FUNCTION_BLOCK TableDeserializer
VAR
	_DataString : POINTER TO STRING;
	dataLength : DINT;
	rowDefinition : __SYSTEM.AnyType;
	_RowCount : DINT;
	_ColumnDefinitionBuffer : ARRAY[0..MaxColumnCount - 1] OF __SYSTEM.AnyType;
	_ColumnNameBuffer : ARRAY[0..MaxColumnCount - 1] OF T_MaxString;
	columnNamesOutput : __SYSTEM.AnyType;
	definedColumns : INT;

	_Separator : STRING := ',';
	_NewLine : STRING := '$N'; // Default is Windows newline.
	_DecimalSeparator : STRING := '.';
END_VAR
VAR CONSTANT
	MaxColumnCount : INT := TableSerializationParameters.DeserializerMaxColumns;
	DefaultDecimalSeparator : STRING := '.';
END_VAR

{attribute 'monitoring' := 'call'}
PROPERTY DataString : POINTER TO STRING
GET
DataString := _DataString;
END_GET
SET
_DataString := DataString;
END_SET
END_PROPERTY

{attribute 'monitoring' := 'call'}
PROPERTY DecimalSeparator : STRING
GET
DecimalSeparator := _DecimalSeparator;
END_GET
SET
_DecimalSeparator := DecimalSeparator;
END_SET
END_PROPERTY

METHOD DefineColumnNamesOutput : REFERENCE TO TableDeserializer
VAR_INPUT
	columnNames : ANY; 
END_VAR
columnNamesOutput := columnNames;

DefineColumnNamesOutput REF= THIS^;
END_METHOD

METHOD DefineNextColumn : REFERENCE TO TableDeserializer
VAR_INPUT
	columnInFirstRow : ANY; 
END_VAR
IF (definedColumns < MaxColumnCount) THEN
	_ColumnDefinitionBuffer[definedColumns] := columnInFirstRow;
	definedColumns := definedColumns + 1;
END_IF

DefineNextColumn REF= THIS^;
END_METHOD

METHOD DefineRow : REFERENCE TO TableDeserializer
VAR_INPUT
	firstRow : ANY;
END_VAR
rowDefinition := firstRow;

DefineRow REF= THIS^;
END_METHOD

METHOD Deserialize : DINT
VAR_INPUT
	includingHeader : BOOL;
END_VAR
VAR
	caret : DINT;
END_VAR
dataLength := TO_DINT(LEN2(dataString));
IF (includingHeader) THEN
	caret := ReadHeader();
END_IF
caret := ReadAllRows(caret);

Deserialize := caret;
END_METHOD

{attribute 'monitoring' := 'call'}
PROPERTY NewLine : STRING
GET
NewLine := _NewLine;
END_GET
SET
_NewLine := NewLine;
END_SET
END_PROPERTY

METHOD PRIVATE ReadAllRows : DINT
VAR_INPUT
	startCaret : DINT;
END_VAR
VAR
	caret : DINT;
	i : DINT;
END_VAR
caret := startCaret;

FOR i := 0 TO _RowCount - 1 DO
	IF (caret >= dataLength) THEN
		EXIT;
	END_IF
	caret := ReadRow(i, caret);
END_FOR

ReadAllRows := caret;
END_METHOD

METHOD PRIVATE ReadHeader : DINT
VAR
	i : DINT;
	
	caret : DINT;
	lineEnd : DINT;
	cellLength : DINT;
	
	cell : T_MaxString;
END_VAR
ClearData(_ColumnNameBuffer);

lineEnd := TO_DINT(FIND2(pSrcString := _DataString, pFindString := ADR(_NewLine)));
IF (lineEnd = 0) THEN
	lineEnd := dataLength;
END_IF

FOR i := 0 TO definedColumns - 1 DO
	cellLength := TO_DINT(FIND2(pSrcString := _DataString + TO_DWORD(caret), pFindString := ADR(_Separator)));
	IF (caret + cellLength > lineEnd) THEN
		cellLength := lineEnd - caret;
	END_IF
	IF (cellLength = 0) THEN
		cellLength := lineEnd;
	END_IF

	MEMSET(destAddr := ADR(cell), fillByte := 0, n := SIZEOF(cell));
	MEMCPY(destAddr := ADR(cell), srcAddr := _DataString + TO_DWORD(caret), n := TO_UDINT(MIN(SIZEOF(cell) - 1, cellLength - 1)));
	StringToAny(cell, _ColumnNameBuffer[i]);
	
	IF (cellLength = dataLength) THEN
		caret := lineEnd;
	ELSIF (cellLength = lineEnd) THEN
		caret := lineEnd;
	ELSE
		caret := caret + cellLength;
	END_IF
END_FOR

MEMCPY(
	destAddr := columnNamesOutput.pValue,
	srcAddr := ADR(_ColumnNameBuffer),
	n := TO_UDINT(MIN(columnNamesOutput.diSize, SIZEOF(_ColumnNameBuffer)))
);

ReadHeader := caret;
END_METHOD

METHOD PRIVATE ReadRow : DINT
VAR_INPUT
	row : DINT;
	startCaret : DINT;
END_VAR
VAR
	i : DINT;
	
	caret : DINT;
	lineLength : DINT;
	cellLength : DINT;
	
	cell : T_MaxString;
	
	tableCell : __SYSTEM.AnyType;
END_VAR
caret := startCaret;

lineLength := TO_DINT(FIND2(pSrcString := _DataString + TO_DWORD(caret), pFindString := ADR(_NewLine)));
IF (lineLength = 0) THEN
	lineLength := dataLength;
END_IF

FOR i := 0 TO definedColumns - 1 DO
  IF (caret >= dataLength) THEN
		EXIT;
	END_IF
	cellLength := TO_DINT(FIND2(pSrcString := _DataString + TO_DWORD(caret), pFindString := ADR(_Separator)));
	IF (cellLength = 0 OR caret + cellLength > startCaret + lineLength) THEN
		cellLength := lineLength + startCaret - caret;
	END_IF
	IF (cellLength = 0) THEN
		caret := dataLength;
		EXIT;
	END_IF

	ClearData(cell);
	MEMCPY(destAddr := ADR(cell), srcAddr := _DataString + TO_DWORD(caret), n := TO_UDINT(MIN(SIZEOF(cell) - 1, cellLength - 1)));
	tableCell := _ColumnDefinitionBuffer[i];
	tableCell.pValue := tableCell.pValue + TO_DWORD(rowDefinition.diSize * row);
	CASE TO_INT(tableCell.TypeClass) OF
		TYPE_REAL, TYPE_LREAL:
			ReplaceString(cell, _DecimalSeparator, DefaultDecimalSeparator);
	END_CASE
	StringToAnyType(cell, tableCell);
	
	IF (cellLength = dataLength) THEN
		caret := startCaret + lineLength;
	ELSIF (cellLength = lineLength) THEN
		caret := startCaret + lineLength;
	ELSE
		caret := caret + cellLength;
	END_IF
END_FOR

ReadRow := caret;
END_METHOD

{attribute 'monitoring' := 'call'}
PROPERTY RowCount : DINT
GET
RowCount := _RowCount;
END_GET
SET
_RowCount := RowCount;
END_SET
END_PROPERTY

{attribute 'monitoring' := 'call'}
PROPERTY Separator : STRING
GET
Separator := _Separator;
END_GET
SET
_Separator := Separator;
END_SET
END_PROPERTY

END_FUNCTION_BLOCK

(* stored: Version 1.1.0.1
   POU TableDeserializer: Id {ac25e541-c19a-0342-2f23-5f00fecd60cf}, SpecialFunc None
   Property DataString: Id {3487dc60-cc91-4a43-8a0d-0551ca27c8b6}
   Get Get: Id {8cc0e152-d7a2-4043-a052-b993cd54d7db}
   Set Set: Id {bd17b9aa-3d4c-41a0-b30b-2c68dc3bad68}
   Property DecimalSeparator: Id {d3dad73a-0f1a-41a0-a71e-05862e1d10d8}
   Get Get: Id {43213d27-d09c-0e10-0860-afcf924a6719}
   Set Set: Id {10f316a8-26b4-0f7b-0428-7a47d65a91e1}
   Method DefineColumnNamesOutput: Id {de401d8b-b754-0646-0d01-b230f4361c5f}
   Method DefineNextColumn: Id {7a1778bf-3544-0497-095c-7861e545f68b}
   Method DefineRow: Id {f358bb43-9e62-0f97-1aa1-51c1ec6b43cf}
   Method Deserialize: Id {469a7f4d-b005-006e-04b0-81df065e5112}
   Property NewLine: Id {e231f9e3-68dc-40f1-baa5-667ee97338a5}
   Get Get: Id {4313d227-83a4-058f-0465-9ca8841186a4}
   Set Set: Id {ada97d3e-dd7f-0ada-0be1-e68f70e46dbd}
   Method ReadAllRows: Id {e19a843a-8d18-0ff9-0de4-c88d595663c8}
   Method ReadHeader: Id {d90cef34-8289-0ac4-2959-a4dd8ac2e400}
   Method ReadRow: Id {9e4c8000-7c69-0be9-232c-fb4179063f04}
   Property RowCount: Id {ed443da8-c273-0153-280d-4c621b350138}
   Get Get: Id {7ad9c8fe-4559-08da-00c7-f01597993e7f}
   Set Set: Id {655700f4-3d23-0ab3-1716-3908da2b156b}
   Property Separator: Id {b68ca63d-6f90-04d5-2320-3780f007dffc}
   Get Get: Id {fce9d174-de86-05b6-20d4-813c0e4499e4}
   Set Set: Id {eaa5df53-009d-0b64-0cef-d74aa32ee656} *)
